// TIA Portal project "guess the number" (V17)

(* hardware
DEVICE "S7-1500/ET200MP station_1"  S7-1500 station
   slot 0: "Rail_0"  Rack  6ES7 590-1***0-0AA0
   slot 1: "PLC_1"  CPU 1512C-1 PN  6ES7 512-1CK00-0AB0  V2.1
      slot 3: "CPU display_1"  6ES7591-1AA00-0AA0
      slot 32768: "PROFINET interface_1"  X1
         slot 32769: "Port_1"  X1 P1
         slot 32770: "Port_2"  X1 P2
*)

// ===== PLC "PLC_1"  CPU 1512C-1 PN =====

VAR_GLOBAL   // PLC tag table "Default tag table"
   "gameOver" AT %I0.0 : Bool;
   "Start" AT %I0.1 : Bool;
   "guess" AT %ID0 : DInt;
   "System_Byte" AT %MB1 : Byte;
   "FirstScan" AT %M1.0 : Bool;
   "DiagStatusUpdate" AT %M1.1 : Bool;
   "AlwaysTRUE" AT %M1.2 : Bool;
   "AlwaysFALSE" AT %M1.3 : Bool;
   "Clock_Byte" AT %MB0 : Byte;
   "Clock_10Hz" AT %M0.0 : Bool;
   "Clock_5Hz" AT %M0.1 : Bool;
   "Clock_2.5Hz" AT %M0.2 : Bool;
   "Clock_2Hz" AT %M0.3 : Bool;
   "Clock_1.25Hz" AT %M0.4 : Bool;
   "Clock_1Hz" AT %M0.5 : Bool;
   "Clock_0.625Hz" AT %M0.6 : Bool;
   "Clock_0.5Hz" AT %M0.7 : Bool;
END_VAR

DATA_BLOCK "Data"   // DB1
{ S7_Optimized_Access := 'TRUE' }
VERSION : 0.1
   VAR
      randomNumber : Int;
      guess : Int;
      gameOver : Bool;
      gameWon : Bool;
      gameLost : Bool;
      RetVal : Int;
      Start : Bool;
      InfoZ : UDInt;
      REST : UDInt;
      timeJETZT : DTL;
   END_VAR
BEGIN
END_DATA_BLOCK

FUNCTION "game" : Void   // FC1, SCL
{ S7_Optimized_Access := 'TRUE' }
VERSION : 0.1
BEGIN

   WHILE "Start" = TRUE DO
       WHILE "gameOver" = FALSE DO
           IF "guess" = "Data".REST THEN
               "Data".gameWon := 1;
               "Data".gameLost := 0;
               "gameOver" := TRUE;
           ELSIF "guess" <> "Data".REST THEN
               "Data".gameLost := 1;
               "Data".gameWon := 0;
           END_IF;
       END_WHILE;

       WHILE "gameOver" = FALSE DO
           "Data".RetVal := RD_SYS_T(OUT => "Data".timeJETZT);
           "Data".InfoZ := "Data".timeJETZT.NANOSECOND / 10000;
           "Data".REST := ("Data".InfoZ MOD 100) + 1;
       END_WHILE;
   END_WHILE;
END_FUNCTION

ORGANIZATION_BLOCK "Main"   // OB1, LAD, ProgramCycle
TITLE = "Main Program Sweep (Cycle)"
{ S7_Optimized_Access := 'TRUE' }
VERSION : 0.1
   VAR_INPUT
      Initial_Call : Bool;   // Initial call of this OB
      Remanence : Bool;   // =True, if remanent data are available
   END_VAR
BEGIN

REGION Network 1
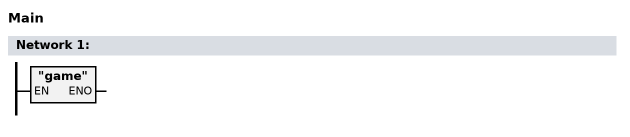
   RUNG wire#powerrail
      "game"()
   END_RUNG
   // the same network as SCL:
   "game"();
END_REGION
END_ORGANIZATION_BLOCK